Fanuc KAREL source: kc00007.KL

-- PROVISIONAL review KL for V770-1; original PC SHA256 4912b7475dc16734b5ce58ca2ed6dbf7aeffca5aede37a405fc52bb2ea336128
-- Incomplete behavior may be omitted. Consult companion uncertainty JSON. Do not deploy.
PROGRAM KC00007
%NOLOCKGROUP
BEGIN
  -- UNRESOLVED_PC offsets 5-51; opcodes 27,22,1C,22,22,22,1C,22,31
  -- UNRESOLVED_PC offsets 56-60; opcodes 7F
END KC00007
